// TIA Portal V16 export
// export: Created 2024-12-03T15:41:45.0255453Z, ExportSetting WithReadOnly, DisplayName Totally Integrated Automation Portal, DisplayVersion V16 Update 6, DisplayName TIA Portal Version Control Interface, DisplayVersion V16 Update 2, DisplayName TIA Portal Openness, DisplayVersion V16 Update 6, DisplayName TIA Portal Teamcenter Gateway, DisplayVersion V16, DisplayName SINAMICS Startdrive Advanced, DisplayVersion V16 Update 5, DisplayName SINAMICS Startdrive G130, G150, S120, S150, SINAMICS MV, S210, DisplayVersion V16 Update 5, DisplayName SINAMICS Startdrive G110M, G120, G120C, G120D, G120P, G115D, DisplayVersion V16 Update 5, DisplayName STEP 7 Professional, DisplayVersion V16 Update 6, DisplayName STEP 7 Safety, DisplayVersion V16, DisplayName WinCC Advanced / Unified PC, DisplayVersion V16 Update 6
TYPE "ConveyLinx_IO_IN_OUT_UDT"
// stored: CreationDate 2021-07-13T07:41:36.2278727Z, InterfaceModifiedDate 2020-08-12T06:14:04.3244967Z, IsConsistent true, LibraryConformanceStatus The object is library-conformant., ModifiedDate 2021-03-27T07:36:39.8028956Z
   STRUCT
      spare : Byte := 16#0;
      Male_Up_Left_Pin_2 : Bool := false;   // Male_Up left pin 2
      Female_Down_Left_Pin_2 : Bool := false;   // Female_Down left pin 2
      Male_Up_Right_Pin_2 : Bool := false;   // Male_Up right pin 2
      Female_Down_Right_Pin_2 : Bool := false;   // Female_Down right pin 2
      Male_Up_Left_Pin_4 : Bool := false;   // Male_Up left pin 4
      Female_Down_Left_Pin_4 : Bool := false;   // Female_Down left pin 4
      Male_Up_Right_Pin_4 : Bool := false;   // Male_Up right pin 4
      Female_Down_Right_Pin_4 : Bool := false;   // Female_Down right pin 4
   END_STRUCT;
END_TYPE
